VISUALIZATION Visualization  // 2x2
END_VISUALIZATION

(* stored: Version 1.1.0.1, ProductVersion 3.1.4024.12
   Visu Visualization: Id {2aa6c8fd-ffdc-46a8-972d-865fa82dc898} *)
